FUNCTION_BLOCK PUBLIC PAEMaterialSensor EXTENDS PAESensorDigital
VAR_INPUT
END_VAR
VAR_OUTPUT
END_VAR
VAR
END_VAR

END_FUNCTION_BLOCK

(* stored: Version 1.1.0.1, ProductVersion 3.1.4020.6
   POU PAEMaterialSensor: Id {c38592fd-363e-4c27-a636-d85c086ca7ba}, SpecialFunc None *)
